// Core §7.7 under test: open-by-default, threshold denial, data-driven login through
// the local provider, secret cleared, logout re-denies, denied attempts audited.
FUNCTION_BLOCK FB_Access_Tests EXTENDS TcUnit.FB_TestSuite
VAR
    _u  : FB_ProbeUnit;
    _pr : FB_LocalAccessProvider;
    _w  : BOOL;
END_VAR

Default_policy_is_fully_open();
Threshold_denies_then_login_permits_then_logout_denies();
Policy_rejects_invalid_ordinals_and_timeout();
Re_registering_replaces_the_PIN();

METHOD Default_policy_is_fully_open
TEST('Default_policy_is_fully_open');
IF NOT _w THEN
    _u.Setup('Test.AccessUnit');
    _pr.Register(User := 'tech1', Pin := '4711', Level := E_AccessLevel.TECHNICIAN);
    _u();                                              // first scan wires audit log
    _u.Access.Setup(Provider := _pr, pAlarmLog := ADR(_u.AlarmLog));
    _w := TRUE;
END_IF
AssertTrue(Condition := _u.Access.Permits(Gate := E_GatedAction.MODE_CHANGE),
           Message := 'NONE thresholds: no login needed (7.7b — the fully-open station)');
AssertTrue(Condition := _u.SetMode(Mode := E_Mode.MANUAL),
           Message := 'mode change works without any session');
AssertTrue(Condition := _u.SetMode(Mode := E_Mode.AUTO), Message := 'back to AUTO');
_u(); _u(); _u();
TEST_FINISHED();
END_METHOD

METHOD Threshold_denies_then_login_permits_then_logout_denies
TEST('Threshold_denies_then_login_permits_then_logout_denies');
_u.Access.ConfigureRequired(Gate := E_GatedAction.MODE_CHANGE, Level := E_AccessLevel.TECHNICIAN);
AssertFalse(Condition := _u.SetMode(Mode := E_Mode.MANUAL),
            Message := 'denied below threshold (7.7c) — PLC re-checks, not the HMI');
AssertTrue(Condition := _u.AlarmLog.RingHead > 0,
           Message := 'denied attempt audited as a MESSAGE event (8.3)');
// wrong PIN
_u.Access.RequestLogin(User := 'tech1', Secret := '0000');
_u();
AssertTrue(Condition := _u.Access.LoginFailed, Message := 'wrong PIN rejected');
AssertEquals_DINT(Expected := TO_DINT(E_AccessLevel.NONE),
                  Actual := TO_DINT(_u.Access.CurrentLevel), Message := 'level stays NONE');
// correct PIN — data-driven login (3.10a')
_u.Access.RequestLogin(User := 'tech1', Secret := '4711');
_u();
AssertEquals_DINT(Expected := TO_DINT(E_AccessLevel.TECHNICIAN),
                  Actual := TO_DINT(_u.Access.CurrentLevel), Message := 'TECHNICIAN session');
AssertEquals_STRING(Expected := '', Actual := _u.Access.ReqSecret,
                    Message := 'secret cleared after the attempt (7.7c)');
AssertTrue(Condition := _u.SetMode(Mode := E_Mode.MANUAL),
           Message := 'permitted at sufficient level');
_u.Access.RequestLogout();
_u();
AssertEquals_DINT(Expected := TO_DINT(E_AccessLevel.NONE),
                  Actual := TO_DINT(_u.Access.CurrentLevel), Message := 'logged out');
AssertFalse(Condition := _u.SetMode(Mode := E_Mode.AUTO),
            Message := 'denied again after logout');
_u.Access.ConfigureRequired(Gate := E_GatedAction.MODE_CHANGE, Level := E_AccessLevel.NONE);  // restore
_u.SetMode(Mode := E_Mode.AUTO);
_u(); _u();
TEST_FINISHED();
END_METHOD

METHOD Policy_rejects_invalid_ordinals_and_timeout
VAR
    invalidGate : E_GatedAction;
    invalidLevel : E_AccessLevel;
END_VAR
TEST('Policy_rejects_invalid_ordinals_and_timeout');
invalidGate := 99;
invalidLevel := 99;
AssertFalse(Condition := _u.Access.ConfigureRequired(
    Gate := invalidGate, Level := E_AccessLevel.ADMIN),
    Message := 'out-of-range gate fails closed');
AssertFalse(Condition := _u.Access.ConfigureRequired(
    Gate := E_GatedAction.DATA_WRITE, Level := invalidLevel),
    Message := 'out-of-range level fails closed');
AssertFalse(Condition := _u.Access.ConfigureSessionTimeout(TimeoutMs := 604800001),
    Message := 'timeout above seven days rejected');
AssertTrue(Condition := _u.Access.ConfigureSessionTimeout(TimeoutMs := 900000),
    Message := 'bounded timeout accepted');
AssertEquals_DINT(Expected := 900000,
    Actual := TIME_TO_DINT(_u.Access.Policy.SessionTimeout),
    Message := 'accepted timeout stored in policy');
_u.Access.ConfigureSessionTimeout(TimeoutMs := 0);
TEST_FINISHED();
END_METHOD

// §14 - the table holds only a salted hash, so the PIN is checked by hashing the
// attempt: the new PIN is accepted, the old one and the hash's own inputs are not.
METHOD Re_registering_replaces_the_PIN
VAR
    p : FB_LocalAccessProvider;
END_VAR
TEST('Re_registering_replaces_the_PIN');
AssertTrue(Condition := p.Register(User := 'op', Pin := '1111', Level := E_AccessLevel.OPERATOR),
    Message := 'registered');
AssertTrue(Condition := p.Register(User := 'eng', Pin := '1111', Level := E_AccessLevel.ENGINEER),
    Message := 'a second user may share the PIN (own salt)');
AssertEquals_DINT(Expected := TO_DINT(E_AccessLevel.OPERATOR),
    Actual := TO_DINT(p.Authenticate(User := 'op', Secret := '1111')), Message := 'op accepted');
AssertEquals_DINT(Expected := TO_DINT(E_AccessLevel.ENGINEER),
    Actual := TO_DINT(p.Authenticate(User := 'eng', Secret := '1111')), Message := 'eng accepted');
AssertTrue(Condition := p.Register(User := 'op', Pin := '2222', Level := E_AccessLevel.OPERATOR),
    Message := 're-registered');
AssertEquals_DINT(Expected := TO_DINT(E_AccessLevel.NONE),
    Actual := TO_DINT(p.Authenticate(User := 'op', Secret := '1111')), Message := 'old PIN refused');
AssertEquals_DINT(Expected := TO_DINT(E_AccessLevel.OPERATOR),
    Actual := TO_DINT(p.Authenticate(User := 'op', Secret := '2222')), Message := 'new PIN accepted');
AssertEquals_DINT(Expected := TO_DINT(E_AccessLevel.NONE),
    Actual := TO_DINT(p.Authenticate(User := 'nobody', Secret := '2222')), Message := 'unknown user refused');
AssertEquals_DINT(Expected := TO_DINT(E_AccessLevel.NONE),
    Actual := TO_DINT(p.Authenticate(User := 'op', Secret := '')), Message := 'empty secret refused');
TEST_FINISHED();
END_METHOD

END_FUNCTION_BLOCK

(* stored: Version 1.1.0.1, ProductVersion 3.1.4024.12
   POU FB_Access_Tests: Id {eaea0db1-5490-46ab-b19f-9e2baa566e81}, SpecialFunc None
   Method Default_policy_is_fully_open: Id {1c4a183c-7370-44bd-8a31-5b4260b328aa}
   Method Threshold_denies_then_login_permits_then_logout_denies: Id {c0445ba8-3700-466b-8cca-5b2681b333bc}
   Method Policy_rejects_invalid_ordinals_and_timeout: Id {306f8d36-b5da-47cb-9e7d-4715429595ce}
   Method Re_registering_replaces_the_PIN: Id {17c6fa1d-6080-41ad-96be-bf1b4a4ceece} *)
